{attribute addProperty BoxType "IODEVICETYPE_ETHERCATPROT"}
{attribute addProperty Id "Term_1_EK1200Term_1_EK1200_134F30391897237.125SyncUnitsSyncUnits_235333EF26032.5InputsInputs_5FC39E3C8010OutputsOutputs_C46FA7B3486InfoDataInfoData_45F98C5022428"}
{attribute addProperty CRC "1974531758"}
{attribute addProperty SizeInBites "2509"}
{attribute addProperty SizeInBytes "313.625"}
TYPE Device_1_EtherCAT_75B0F6AE :
STRUCT
	{attribute addProperty Name "Term_1_EK1200"}
	Term_1_EK1200 : Term_1_EK1200_134F3039;
	{attribute addProperty Name "SyncUnits"}
	SyncUnits : SyncUnits_235333EF;
	{attribute addProperty Name "Inputs"}
	Inputs : Inputs_5FC39E3C;
	{attribute addProperty Name "Outputs"}
	Outputs : Outputs_C46FA7B3;
	{attribute addProperty Name "InfoData"}
	InfoData : InfoData_45F98C50;
END_STRUCT
END_TYPE

(* stored: Version 1.2.0.0, ProductVersion 3.1.4024.9
   DUT Device_1_EtherCAT_75B0F6AE: Id {261ae2bb-dad4-0470-2875-ac93148f53c3} *)
